TYPE ST_FanucCNCEventSourceDetails :
STRUCT
	MainType : BYTE;
	SubType : BYTE;
	CNCNo : BYTE;
	PathNo : BYTE;
END_STRUCT
END_TYPE

(* stored: Version 1.1.0.1, ProductVersion 3.1.4024.12
   DUT ST_FanucCNCEventSourceDetails: Id {ee0b50fa-bc9a-4945-8ed3-a83357c3fd9d} *)
